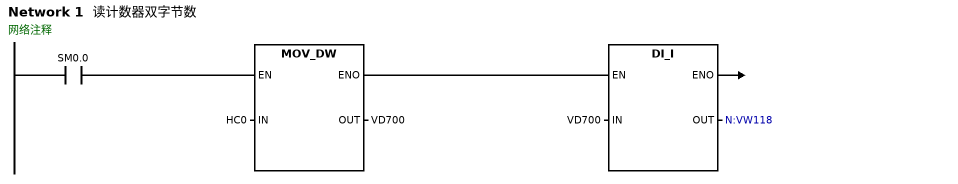
[picture p24: INT1 networks 1-1]
Network 1 // 读计数器双字节数
// 网络注释
LD     SM0.0
MOVD   HC0, VD700
AENO
DTI    VD700, N:VW118
END_INTERRUPT_BLOCK

DATA_BLOCK_TAB 数据块
BEGIN
//数据块注释
//按F1获得帮助和范例数据块
//BEGIN TD200_BLOCK ----------------------------
VB0      'TD'
VB2      16#60               //将“语言”设为中文，将“更新”设为尽快 
VB3      16#F0               //将显示设为20字符模式；“向上”键V3.2；“向下”键V3.3；
VB4      1                   //设置讯息数目
VB5      0                   //将功能键通知位设为M0.0 - M0.7
VW6      34                  //将讯息起始地址设为VW34 
VW8      14                  //将讯息启用位起始地址设为VW14 
VW10     0                   //全局密码（如启用）
VW12     256                 //字符集 = 简体中文 
//MESSAGE 1	
//讯息启用位V14.7 
VB34     '                    '
//END TD200_BLOCK ------------------------------
END_DATA_BLOCK_TAB
